PROGRAM DAS_CoreSys
VAR
    UserModeCofig  : PML_UnitModeConfig; //User can configure his own Mode
    MachineControl : FB_MachineControl;
	CoreSys_Stop : BOOL;
	CoreSys_Reset :BOOL;
	CoreSys_Start : BOOL;
	CoreSys_Estop : BOOL;
	OP_Mode : E_UnitMode := E_UnitMode.Manual;
END_VAR

A00_BasicUnit();
A10_StatusCtrl();


CASE GVL_ADS.MachineMode.TargetMode OF
		E_MachineMode.MANUAL:
			OP_Mode := E_UnitMode.Manual;
		E_MachineMode.AUTO:
			OP_Mode := E_UnitMode.Auto;
ELSE
	OP_Mode := E_UnitMode.Manual;
END_CASE
IF OP_Mode = E_UnitMode.Manual THEN
	GVL_ADS.MachineMode.CurrentMode := E_MachineMode.MANUAL;
ELSIF OP_Mode = E_UnitMode.Auto THEN
	GVL_ADS.MachineMode.CurrentMode := E_MachineMode.AUTO;
END_IF

ACTION A00_BasicUnit:
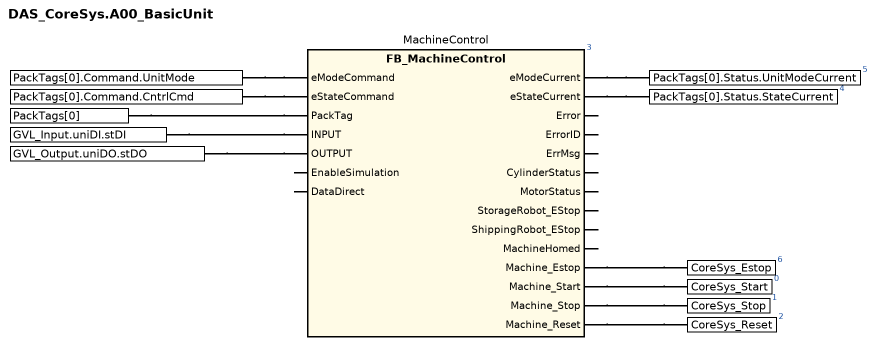
CoreSys_Start := MachineControl.Machine_Start;
CoreSys_Stop := MachineControl.Machine_Stop;
CoreSys_Reset := MachineControl.Machine_Reset;
MachineControl(
    eModeCommand := PackTags[0].Command.UnitMode,
    eStateCommand := PackTags[0].Command.CntrlCmd,
    PackTag := PackTags[0],
    INPUT := GVL_Input.uniDI.stDI,
    OUTPUT := GVL_Output.uniDO.stDO); // FB_MachineControl
PackTags[0].Status.StateCurrent := MachineControl.eStateCurrent;
PackTags[0].Status.UnitModeCurrent := MachineControl.eModeCurrent;
CoreSys_Estop := MachineControl.Machine_Estop;
END_ACTION

ACTION A01_UnitModeConfig:
//UserModeCofig(
//	eMode							:= ePMLUnitMode_Service, 
//	bDisableClearing				:= TRUE, 
//	bDisableStarting				:= TRUE, 
//	bDisableSuspended				:= FALSE, 
//	bDisableStopping				:= TRUE, 
//	bDisableAborting				:= TRUE, 
//	bDisableHolding					:= TRUE, 
//	bDisableHeld					:= TRUE, 
//	bDisableUnholding				:= TRUE, 
//	bDisableSuspending				:= TRUE, 
//	bDisableUnsuspending			:= TRUE, 
//	bDisableResetting				:= TRUE, 
//	bDisableIdle					:= TRUE, 
//	bDisableCompleting				:= TRUE, 
//	bDisableComplete				:= TRUE, 
//	bEnableUnitModeChangeStopped	:= TRUE, 
//	bEnableUnitModeChangeIdle		:= FALSE, 
//	bEnableUnitModeChangeSuspended	:= FALSE, 
//	bEnableUnitModeChangeExecute	:= FALSE, 
//	bEnableUnitModeChangeAborted	:= TRUE, 
//	bEnableUnitModeChangeHeld		:= FALSE, 
//	bEnableUnitModeChangeComplete	:= FALSE, 
//	bError							=> , 
//	nErrorId						=> );
END_ACTION

ACTION A10_StatusCtrl:
IF PackTags[0].Status.UnitModeCurrent = E_UnitMode.Manual THEN
	IF PackTags[0].Status.StateCurrent = ePMLState_Aborted AND NOT MachineControl.Error THEN
		PackTags[0].Command.CntrlCmd := ePMLCommand_Clear;
	END_IF
	IF PackTags[0].Status.StateCurrent = ePMLState_Stopped THEN
		IF OP_Mode = E_UnitMode.Manual THEN
		PackTags[0].Command.CntrlCmd := ePMLCommand_Reset;
		END_IF
	END_IF
	IF PackTags[0].Status.StateCurrent = ePMLState_Idle THEN
		PackTags[0].Command.CntrlCmd := ePMLCommand_Start;
	END_IF
ELSIF PackTags[0].Status.UnitModeCurrent = E_UnitMode.Auto THEN
	IF PackTags[0].Status.StateCurrent = ePMLState_Aborted AND NOT MachineControl.Error THEN
		PackTags[0].Command.CntrlCmd := ePMLCommand_Clear;
	END_IF
	IF PackTags[0].Status.StateCurrent = ePMLState_Stopped THEN
		IF OP_Mode = E_UnitMode.Auto THEN
		PackTags[0].Command.CntrlCmd := ePMLCommand_Reset;
		END_IF
	END_IF
	IF PackTags[0].Status.StateCurrent = ePMLState_Idle THEN
		PackTags[0].Command.CntrlCmd := ePMLCommand_Start;
	END_IF
END_IF

IF PackTags[0].Status.UnitModeCurrent = E_UnitMode.Manual THEN
    IF ((PackTags[0].Status.StateCurrent = ePMLState_Stopped) OR
        (PackTags[0].Status.StateCurrent = ePMLState_Aborted) OR
        (PackTags[0].Status.StateCurrent = ePMLState_Execute)) AND
        MachineControl.MachineHomed
        THEN
        IF OP_Mode = E_UnitMode.Auto THEN
            PackTags[0].Command.UnitMode := E_UnitMode.Auto;
			IF PackTags[0].Status.StateCurrent = ePMLState_Execute THEN
				PackTags[0].Command.CntrlCmd := ePMLCommand_Stop;
			END_IF
        END_IF
    END_IF
ELSIF PackTags[0].Status.UnitModeCurrent = E_UnitMode.Auto THEN
    IF ((PackTags[0].Status.StateCurrent = ePMLState_Stopped) OR
        (PackTags[0].Status.StateCurrent = ePMLState_Aborted) OR
        (PackTags[0].Status.StateCurrent = ePMLState_Execute))
        THEN
        IF OP_Mode = E_UnitMode.Manual THEN
			IF PackTags[0].Status.StateCurrent <> ePMLState_Aborted OR PackTags[0].Status.StateCurrent <> ePMLState_Aborting THEN
				PackTags[0].Command.CntrlCmd := ePMLCommand_Abort;
			END_IF
            PackTags[0].Command.UnitMode := E_UnitMode.Manual;
        END_IF
    END_IF
END_IF

GVL_ADS.OpPannel_Status.EStopBtnStatus := CoreSys_Estop;
GVL_ADS.OpPannel_Status.ResetBtnStatus := CoreSys_Reset;
GVL_ADS.OpPannel_Status.StartBtnStatus := CoreSys_Start;
GVL_ADS.OpPannel_Status.StopBtnStatus := CoreSys_Stop;
// Start
IF PackTags[0].Status.UnitModeCurrent = E_UnitMode.Auto THEN
	CASE PackTags[0].Status.StateCurrent OF
		ePMLState_Idle:
			IF CoreSys_Start THEN
				PackTags[0].Command.CntrlCmd := ePMLCommand_Start;
			END_IF
	END_CASE
END_IF

// Reset & Clear

IF PackTags[0].Status.UnitModeCurrent = E_UnitMode.Auto THEN
	CASE PackTags[0].Status.StateCurrent OF
		ePMLState_Stopped,ePMLState_Complete:
			IF CoreSys_Reset THEN
				PackTags[0].Command.CntrlCmd := ePMLCommand_Reset;
			END_IF
		ePMLState_Aborted:
			IF CoreSys_Reset THEN
				PackTags[0].Command.CntrlCmd := ePMLCommand_Clear;
			END_IF
		ePMLState_Held:
			IF CoreSys_Reset THEN
				PackTags[0].Command.CntrlCmd := ePMLCommand_Unhold;
			END_IF
		ePMLState_Suspended:
			IF CoreSys_Reset THEN
				PackTags[0].Command.CntrlCmd := ePMLCommand_Unsuspend;
			END_IF
	END_CASE
END_IF

// Stop

//IF PackTags[0].Status.UnitModeCurrent = E_UnitMode.Auto THEN
//	CASE PackTags[0].Status.StateCurrent OF
//		ePMLState_Execute:
//			IF CoreSys_Stop THEN
//				PackTags[0].Command.CntrlCmd := ePMLCommand_Suspend;
//			END_IF
//	END_CASE
//END_IF
END_ACTION

END_PROGRAM

(* stored: Version 1.1.0.1, ProductVersion 3.1.4024.13
   POU DAS_CoreSys: Id {e9b99700-e313-4a8f-8c69-88bfc3821eb9}, SpecialFunc None
   Action A00_BasicUnit: Id {c7e27475-5ad9-412e-a816-e24e2a796347}
   Action A01_UnitModeConfig: Id {22b649e9-a085-4601-8ad9-54522ade47b0}
   Action A10_StatusCtrl: Id {10028502-aeef-4c40-8f3a-b78ff76edf33} *)
